(*
Enables pairing with receivers and casting to `I_Component`, but no emitting.
*)
INTERFACE I_Signal EXTENDS I_Debug, I_RawComponent

(*
Pairs the signal with a receiver.  
Returns:
- `Ok` - If pairing is successful.
- `Err.Itf0` - If the receiver interface is invalid.
- `Err.IncArg` - If the `I_Receiver` is invalid.
- `Err.ItfEq` - If the `I_Receiver` is already paired with this `I_Signal`.
- `Err.Ovf` - If there is no space for another pairing.
*)
METHOD Pair : Result
VAR_INPUT
	iReceiver		: I_Receiver;
END_VAR
END_METHOD

PROPERTY Tag : I_Tag
GET
END_GET
END_PROPERTY

(*
Unpairs the signal from a specified receiver.
Returns:
- `Ok` - If unpairing is successful.
- `Err.Itf0` - If the receiver interface is invalid.
- `Err.IncArg` - If the `I_Receiver` is invalid.
- `Err.NoMatch` - If `I_Signal` is not paired with this `I_Receiver`.
*)
METHOD Unpair : Result
VAR_INPUT
	iReceiver		: I_Receiver;
END_VAR
END_METHOD

END_INTERFACE

(* stored: Version 1.1.0.1
   Itf I_Signal: Id {24f70e98-e98e-42d2-be1a-1b78aa21ba77}
   Method Pair: Id {ca87eecf-5514-49b6-9ee7-6f01e2786d2f}
   Property Tag: Id {f8beb40e-c291-4966-b394-9538a673d0a5}
   Get Get: Id {d48c0a70-e0f2-4140-b485-73acb69dfea2}
   Method Unpair: Id {fa23d0f6-12ae-44be-a780-a181f4365fc2} *)
